{attribute 'qualified_only'}
{attribute 'strict'}
TYPE E_DriveLedState :
(
	NotReady := 0,
	Ready	 := 1,
	Running	 := 2,
	Fault    := 3
);
END_TYPE

(* stored: Version 1.1.0.1, ProductVersion 3.1.4024.15
   DUT E_DriveLedState: Id {edd31590-3bc2-4499-b1b4-95cb1d25c38c} *)
